FUNCTION_BLOCK NumericDatatype_TestSuite EXTENDS TcUnit.FB_TestSuite
VAR
END_VAR

TestAddress();
TestClearReference();
TestClone();
TestTypeNameReturnsExpected();
TestIsFloat();
TestIsSigned();
TestMakeReferenceToFollowsReference();
TestMakeReferenceToUpdatesReference();
TestSize();
TestValueReturnsExpectedAfterInit();
TestValueReturnsExpectedAfterChange();
TestSerializeTypeWith();
TestSerializeWith();
TestTryDeserializeFrom();
TestTryMakeReferenceToFollowsReference();
TestTryMakeReferenceToUpdatesReference();

METHOD PUBLIC TestAddress
VAR
    _type : MockNumericDatatype_INT(0);
    notExpected : PVOID := 0;
    actual : PVOID;
END_VAR
TEST('TestAddress');

actual := _type.Address;

AssertFalse(
    Condition := (notExpected = actual),
    Message := 'Type did not return a valid address.'
);

TEST_FINISHED();
END_METHOD

METHOD PUBLIC TestClearReference
VAR
    _type : MockNumericDatatype_INT(0);
	target : INT := 0;
    expected : INT := 0;
    actual : INT;
END_VAR
TEST('TestClearReference');

_type.MakeReferenceTo(target);
_type.ClearReference();
target := 123;

actual := _type.Value;

AssertEquals(
    Expected := expected,
    Actual := actual,
    Message := 'Value did not follow target change'
);

TEST_FINISHED();
END_METHOD

METHOD PUBLIC TestClone
VAR
    _type : MockNumericDatatype_INT(123);
	clone : I_Datatype;
	isValidClone : BOOL;
	compareResult : DINT;
END_VAR
TEST('TestClone');

clone := _type.Clone();

isValidClone := clone <> 0;

IF isValidClone THEN
	compareResult := memcmp(_type.Address, clone.Address, clone.Size);
END_IF

AssertTrue(
	Condition := isValidClone,
	Message := 'Clone did not produce a clone'
);

AssertEquals_DINT(
	Expected := 0,
    Actual := compareResult,
    Message := 'Clone did not return a valid clone.'
);

clone.Dispose();

TEST_FINISHED();
END_METHOD

METHOD PUBLIC TestIsFloat
VAR
    _type : _DWORD(0);
END_VAR
TEST('TestIsFloat');

AssertFalse(
	Condition := _type.IsFloat,
    Message := 'Type did not correctly identify itself as being unsigned'
);

TEST_FINISHED();
END_METHOD

METHOD PUBLIC TestIsSigned
VAR
    _type : MockNumericDatatype_INT(0);
END_VAR
TEST('TestIsSigned');

AssertTrue(
	Condition := _type.IsSigned,
    Message := 'Type did not correctly identify itself as being signed'
);

TEST_FINISHED();
END_METHOD

METHOD PUBLIC TestMakeReferenceToFollowsReference
VAR
    _type : MockNumericDatatype_INT(0);
	target : INT := 0;
    expected : INT := 123;
    actual : INT;
END_VAR
TEST('TestMakeReferenceToFollowsReference');

_type.MakeReferenceTo(target);
target := 123;

actual := _type.Value;

AssertEquals(
    Expected := expected,
    Actual := actual,
    Message := 'Value did not follow target change'
);

TEST_FINISHED();
END_METHOD

METHOD PUBLIC TestMakeReferenceToUpdatesReference
VAR
    _type : MockNumericDatatype_INT(0);
	target : INT := 0;
    expected : INT := 123;
    actual : INT;
END_VAR
TEST('TestMakeReferenceToUpdatesReference');

_type.MakeReferenceTo(target);
_type.Value := 123;

actual := target;

AssertEquals(
    Expected := expected,
    Actual := actual,
    Message := 'Value did not update target'
);

TEST_FINISHED();
END_METHOD

METHOD PUBLIC TestSerializeTypeWith
VAR
    _type : MockNumericDatatype_INT(0);
    serializer : JsonSerializer;
    expected : STRING(500) := '{"typeName":"INT","minValue":-32768,"maxValue":32767,"isSigned":true,"isFloat":false}';
    actual : STRING(500);
END_VAR
TEST('TestSerializeTypeWith');

serializer.Reset();
_type.SerializeTypeWith(serializer);
serializer.TryGetSerializedData(ADR(actual), SIZEOF(actual));

AssertEquals_STRING(
    Expected := expected,
    Actual := actual,
    Message := 'Serialization of type did not return correct string.'
);

TEST_FINISHED();
END_METHOD

METHOD PUBLIC TestSerializeWith
VAR
    _type : MockNumericDatatype_INT(32767);
    serializer : JsonSerializer;
    expected : STRING := '32767';
    actual : STRING(500);
END_VAR
TEST('TestSerializeWith');

serializer.Reset();
_type.SerializeWith(serializer);
serializer.TryGetSerializedData(ADR(actual), SIZEOF(actual));

AssertEquals_STRING(
    Expected := expected,
    Actual := actual,
    Message := 'Serialization of type data did not return correct string.'
);

TEST_FINISHED();
END_METHOD

METHOD PUBLIC TestSize
VAR
    _type : MockNumericDatatype_INT(0);
    expected : UDINT := SIZEOF(INT);
    actual : UDINT;
END_VAR
TEST('TestSize');

actual := _type.Size;

AssertEquals_UDINT(
    Expected := Expected,
    Actual := actual,
    Message := 'Type did not return the correct size.'
);

TEST_FINISHED();
END_METHOD

METHOD PUBLIC TestTryDeserializeFrom
VAR
    deserializer : JsonDeserializer;
    feedback : DeserializerFeedback;
    json : STRING := '32767';
    _type : MockNumericDatatype_INT(0);
    expected : INT := 32767;
    actual : INT;
 END_VAR
TEST('TestTryDeserializeFrom');

deserializer.Reset();
deserializer.TryLoad(json);
_type.TryDeserializeFrom(Deserializer, Feedback);

actual := _type.Value;

AssertEquals(
    Expected := expected,
    Actual := actual,
    Message := 'Type did not deserialize correctly.'
);

TEST_FINISHED();
END_METHOD

METHOD PUBLIC TestTryMakeReferenceToFollowsReference
VAR
    _type : MockNumericDatatype_INT(0);
	target : MockNumericDatatype_INT(0);
    expected : INT := 123;
    actual : INT;
END_VAR
TEST('TestTryMakeReferenceToFollowsReference');

_type.TryMakeReferenceTo(target);
target.Value := 123;

actual := _type.Value;

AssertEquals(
    Expected := expected,
    Actual := actual,
    Message := 'Value did not follow target change'
);

TEST_FINISHED();
END_METHOD

METHOD PUBLIC TestTryMakeReferenceToUpdatesReference
VAR
    _type : MockNumericDatatype_INT(0);
	target : MockNumericDatatype_INT(0);
    expected : INT := 123;
    actual : INT;
END_VAR
TEST('TestTryMakeReferenceToUpdatesReference');

_type.TryMakeReferenceTo(target);
_type.Value := 123;

actual := target.Value;

AssertEquals(
    Expected := expected,
    Actual := actual,
    Message := 'Value did not update target'
);

TEST_FINISHED();
END_METHOD

METHOD PUBLIC TestTypeNameReturnsExpected
VAR
    _type : MockNumericDatatype_INT(0);
    expected : STRING := 'INT';
    actual : STRING;
END_VAR
TEST('TestTypeNameReturnsExpected');

actual := _type.TypeName;

AssertEquals_STRING(
    Expected := expected,
    Actual := actual,
    Message := 'Type did not return correct iec type.'
);

TEST_FINISHED();
END_METHOD

METHOD PUBLIC TestValueReturnsExpectedAfterChange
VAR
    _type : MockNumericDatatype_INT(0);
    expected : INT := 32767;
    actual : INT;
END_VAR
TEST('TestValueReturnsExpectedAfterChange');

_type.Value := 32767;

actual := _type.Value;

AssertEquals(
    Expected := expected,
    Actual := actual,
    Message := 'Expected value not returned after change.'
);

TEST_FINISHED();
END_METHOD

METHOD PUBLIC TestValueReturnsExpectedAfterInit
VAR
    _type : MockNumericDatatype_INT(32767);
    expected : INT := 32767;
    actual : INT;
END_VAR
TEST('TestValueReturnsExpectedAfterInit');

actual := _type.Value;

AssertEquals(
    Expected := expected,
    Actual := actual,
    Message := 'Expected value not returned after Init.'
);

TEST_FINISHED();
END_METHOD

END_FUNCTION_BLOCK

(* stored: Version 1.1.0.1, ProductVersion 3.1.4024.12
   POU NumericDatatype_TestSuite: Id {96a7ab73-a913-4f8e-8a2f-3ed98c4fdc93}, SpecialFunc None
   Method TestAddress: Id {ab8adec7-0eaf-422a-af2c-f5b93eec3375}
   Method TestClearReference: Id {02641ec5-640c-02a6-0764-dca1ba33095a}
   Method TestClone: Id {36e8ef9c-47ae-077c-3382-48fd5378a88a}
   Method TestIsFloat: Id {b63a6895-720b-49eb-99ff-ca044c3d33a2}
   Method TestIsSigned: Id {378dc2a1-16db-0f08-2f72-db867898717d}
   Method TestMakeReferenceToFollowsReference: Id {edd879ed-8ec6-0727-1d2a-b292e4382fa3}
   Method TestMakeReferenceToUpdatesReference: Id {83845776-c6e3-0354-2435-b91da0e9df04}
   Method TestSerializeTypeWith: Id {32ad0aa1-be6a-42cf-aaa7-bc7b586be18e}
   Method TestSerializeWith: Id {887ce0e9-89b2-49be-bcc9-511505717dee}
   Method TestSize: Id {72df271b-2e7d-411f-9e36-9c9bc4e5c76a}
   Method TestTryDeserializeFrom: Id {1eae0fc6-1ebe-4bbb-8c2d-d9dc7cb42ac5}
   Method TestTryMakeReferenceToFollowsReference: Id {a83e39a5-9126-0c0b-3741-132358e1880a}
   Method TestTryMakeReferenceToUpdatesReference: Id {4d80e395-74dc-0585-020b-0d31aea195f6}
   Method TestTypeNameReturnsExpected: Id {4f1f55dc-8b36-4c30-9c88-d7c35fd32871}
   Method TestValueReturnsExpectedAfterChange: Id {e4687985-10d0-46c6-b218-2c645518b0d7}
   Method TestValueReturnsExpectedAfterInit: Id {9fa13c26-a280-4a61-8071-453a98178d49} *)
